// TIA Portal V17 export
// export: Created 2022-07-20T07:02:37.1953579Z, ExportSetting WithDefaults, DisplayName Totally Integrated Automation Portal, DisplayVersion V17, DisplayName TIA Portal Openness, DisplayVersion V17, DisplayName TIA Portal Version Control Interface, DisplayVersion V17, DisplayName SINAMICS Startdrive Advanced, DisplayVersion V17, DisplayName SINAMICS Startdrive G130, G150, S120, S150, SINAMICS MV, S210, DisplayVersion V17, DisplayName SINAMICS Startdrive G110M, G120, G120C, G120D, G120P, G115D, DisplayVersion V17, DisplayName STEP 7 Professional, DisplayVersion V17, DisplayName STEP 7 Safety, DisplayVersion V17, DisplayName WinCC Advanced, DisplayVersion V17
VAR_GLOBAL   // PLC tag table "Printer_P2_Vertical_Motor_Headstray_Lexium_CommunicationTable"
   Printer_P2_Vertical_Motor_Headstray_Lexium_MotorDataInput AT %I52.0 : "TLexium_MDrv_Drv2Plc";
   Printer_P2_Vertical_Motor_Headstray_Lexium_MotorDataOutput AT %Q40.0 : "TLexium_MDrv_Plc2Drv";
END_VAR
